FUNCTION DWORD_TO_BOOLS
  (* Standard: 61499-1 *)
  (* Version 1.0, 2024-02-22, franz *)
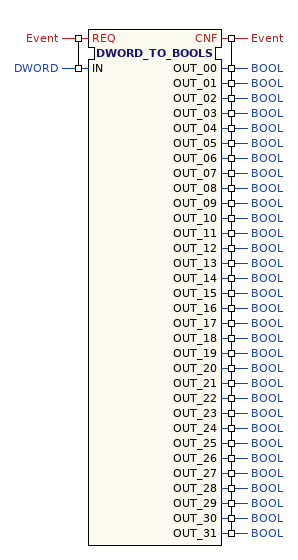
  EVENT_INPUT
    REQ WITH IN; (* Normal Execution Request *)
  END_EVENT
  EVENT_OUTPUT
    CNF WITH OUT_00, OUT_01, OUT_02, OUT_03, OUT_04, OUT_05, OUT_06, OUT_07, OUT_08, OUT_09, OUT_10, OUT_11, OUT_12, OUT_13, OUT_14, OUT_15, OUT_16, OUT_17, OUT_18, OUT_19, OUT_20, OUT_21, OUT_22, OUT_23, OUT_24, OUT_25, OUT_26, OUT_27, OUT_28, OUT_29, OUT_30, OUT_31; (* Execution Confirmation *)
  END_EVENT
  VAR_INPUT
    IN : DWORD; (* DWORD Input *)
  END_VAR
  VAR_OUTPUT
    OUT_00 : BOOL; (* BIT 00 *)
    OUT_01 : BOOL; (* BIT 01 *)
    OUT_02 : BOOL; (* BIT 02 *)
    OUT_03 : BOOL; (* BIT 03 *)
    OUT_04 : BOOL; (* BIT 04 *)
    OUT_05 : BOOL; (* BIT 05 *)
    OUT_06 : BOOL; (* BIT 06 *)
    OUT_07 : BOOL; (* BIT 07 *)
    OUT_08 : BOOL; (* BIT 08 *)
    OUT_09 : BOOL; (* BIT 09 *)
    OUT_10 : BOOL; (* BIT 10 *)
    OUT_11 : BOOL; (* BIT 11 *)
    OUT_12 : BOOL; (* BIT 12 *)
    OUT_13 : BOOL; (* BIT 13 *)
    OUT_14 : BOOL; (* BIT 14 *)
    OUT_15 : BOOL; (* BIT 15 *)
    OUT_16 : BOOL; (* BIT 16 *)
    OUT_17 : BOOL; (* BIT 17 *)
    OUT_18 : BOOL; (* BIT 18 *)
    OUT_19 : BOOL; (* BIT 19 *)
    OUT_20 : BOOL; (* BIT 20 *)
    OUT_21 : BOOL; (* BIT 21 *)
    OUT_22 : BOOL; (* BIT 22 *)
    OUT_23 : BOOL; (* BIT 23 *)
    OUT_24 : BOOL; (* BIT 24 *)
    OUT_25 : BOOL; (* BIT 25 *)
    OUT_26 : BOOL; (* BIT 26 *)
    OUT_27 : BOOL; (* BIT 27 *)
    OUT_28 : BOOL; (* BIT 28 *)
    OUT_29 : BOOL; (* BIT 29 *)
    OUT_30 : BOOL; (* BIT 30 *)
    OUT_31 : BOOL; (* BIT 31 *)
  END_VAR
  BODY IN ST:
FUNCTION DWORD_TO_BOOLS

VAR_INPUT
	IN : DWORD;    // DWORD Input
END_VAR

VAR_OUTPUT
	OUT_00 : BOOL;    // BIT 00
	OUT_01 : BOOL;    // BIT 01
	OUT_02 : BOOL;    // BIT 02
	OUT_03 : BOOL;    // BIT 03
	OUT_04 : BOOL;    // BIT 04
	OUT_05 : BOOL;    // BIT 05
	OUT_06 : BOOL;    // BIT 06
	OUT_07 : BOOL;    // BIT 07
	OUT_08 : BOOL;    // BIT 08
	OUT_09 : BOOL;    // BIT 09
	OUT_10 : BOOL;    // BIT 10
	OUT_11 : BOOL;    // BIT 11
	OUT_12 : BOOL;    // BIT 12
	OUT_13 : BOOL;    // BIT 13
	OUT_14 : BOOL;    // BIT 14
	OUT_15 : BOOL;    // BIT 15
	OUT_16 : BOOL;    // BIT 16
	OUT_17 : BOOL;    // BIT 17
	OUT_18 : BOOL;    // BIT 18
	OUT_19 : BOOL;    // BIT 19
	OUT_20 : BOOL;    // BIT 20
	OUT_21 : BOOL;    // BIT 21
	OUT_22 : BOOL;    // BIT 22
	OUT_23 : BOOL;    // BIT 23
	OUT_24 : BOOL;    // BIT 24
	OUT_25 : BOOL;    // BIT 25
	OUT_26 : BOOL;    // BIT 26
	OUT_27 : BOOL;    // BIT 27
	OUT_28 : BOOL;    // BIT 28
	OUT_29 : BOOL;    // BIT 29
	OUT_30 : BOOL;    // BIT 30
	OUT_31 : BOOL;    // BIT 31
END_VAR

(* this Function extracts the 32 BOOLS from a dword *)
OUT_00 := IN.0;
OUT_01 := IN.1;
OUT_02 := IN.2;
OUT_03 := IN.3;
OUT_04 := IN.4;
OUT_05 := IN.5;
OUT_06 := IN.6;
OUT_07 := IN.7;
OUT_08 := IN.8;
OUT_09 := IN.9;
OUT_10 := IN.10;
OUT_11 := IN.11;
OUT_12 := IN.12;
OUT_13 := IN.13;
OUT_14 := IN.14;
OUT_15 := IN.15;
OUT_16 := IN.16;
OUT_17 := IN.17;
OUT_18 := IN.18;
OUT_19 := IN.19;
OUT_20 := IN.20;
OUT_21 := IN.21;
OUT_22 := IN.22;
OUT_23 := IN.23;
OUT_24 := IN.24;
OUT_25 := IN.25;
OUT_26 := IN.26;
OUT_27 := IN.27;
OUT_28 := IN.28;
OUT_29 := IN.29;
OUT_30 := IN.30;
OUT_31 := IN.31;
END_FUNCTION
  END_BODY
END_FUNCTION
